(* PLC project TestProject.project, CODESYS CODESYS V3.5 SP16 *)
(* stored: creationDateTime 2020-05-25T13:06:30.288415, modificationDateTime 2020-05-25T13:05:00.4147267 *)

PROGRAM PLC_PRG
  VAR
    mail_arr : ARRAY[1..10] OF STRING := ['Kabanbay', 'Abay', 'Turan', 'Saryarka', 'Pushkina', 'Zeinull', 'Tolegen', 'Hodzhan', 'Zholam', 'Halak'];
    Reader : BarCodeReader;
    i : INT;
  END_VAR

                    IF Start THEN
WHILE TRUE DO
	Timer1(IN:= NOT Timer1.Q AND Start,  PT:=T#2s);
	IF Timer1.Q THEN
		Reader(mail_address:=mail_arr[i]);
		i:=i+1;
	END_IF
END_WHILE
END_IF


                  
END_PROGRAM

FUNCTION_BLOCK BarCodeReader
  VAR_INPUT
    mail_address : STRING;
  END_VAR
  VAR_OUTPUT
    box_num : INT;
  END_VAR
  VAR
    TimerK : TON;
  END_VAR

                    IF  LEFT(mail_address,1)>='A' AND LEFT(mail_address,1)<'F' THEN
	Position_x := 0;
	Position_y := 0;
	IF box1full THEN
		REPEAT
			TimerK(IN:= NOT TimerK.Q,  PT:=T#650MS);
			IF TimerK.Q AND Start THEN
				Position_x:=Position_x+155;
			END_IF
		UNTIL Position_x = 1550
		END_REPEAT
		Position_y:= 150;
		storage:=storage+1;
	ELSE
		REPEAT
			TimerK(IN:= NOT TimerK.Q,  PT:=T#500MS);
			IF TimerK.Q AND Start THEN
				Position_x:=Position_x+67;
			END_IF
		UNTIL Position_x = 335
		END_REPEAT
		Position_y:= 150;
		let1:=let1+1;
	END_IF
	
ELSIF LEFT(mail_address,1)>='F' AND LEFT(mail_address,1)<'K' THEN
	Position_x := 0;
	Position_y := 0;
	IF box2full THEN
		REPEAT
			TimerK(IN:= NOT TimerK.Q,  PT:=T#650MS);
			IF TimerK.Q AND Start THEN
				Position_x:=Position_x+155;
			END_IF
		UNTIL Position_x = 1550
		END_REPEAT
		Position_y:= 150;
		storage:=storage+1;
	ELSE
		REPEAT
			TimerK(IN:= NOT TimerK.Q,  PT:=T#500MS);
			IF TimerK.Q AND Start THEN
				Position_x:=Position_x+55;
			END_IF
		UNTIL Position_x = 550
		END_REPEAT
		Position_y:= 150;
		let2:=let2+1;
	END_IF

ELSIF LEFT(mail_address,1)>='K' AND LEFT(mail_address,1)<'P' THEN
	Position_x := 0;
	Position_y := 0;
	IF box3full THEN
		REPEAT
			TimerK(IN:= NOT TimerK.Q,  PT:=T#650MS);
			IF TimerK.Q AND Start THEN
				Position_x:=Position_x+155;
			END_IF
		UNTIL Position_x = 1550
		END_REPEAT
		Position_y:= 150;
		storage:=storage+1;
	ELSE
		REPEAT
			TimerK(IN:= NOT TimerK.Q,  PT:=T#600MS);
			IF TimerK.Q AND Start THEN
				Position_x:=Position_x+107;
			END_IF
		UNTIL Position_x = 749
		END_REPEAT
		Position_y:= 150;
		let3:=let3+1;
	END_IF

ELSIF LEFT(mail_address,1)>='P' AND LEFT(mail_address,1)<'U' THEN
	Position_x := 0;
	Position_y := 0;
	IF box4full THEN
		REPEAT
			TimerK(IN:= NOT TimerK.Q,  PT:=T#650MS);
			IF TimerK.Q AND Start THEN
				Position_x:=Position_x+155;
			END_IF
		UNTIL Position_x = 1550
		END_REPEAT
		Position_y:= 150;
		storage:=storage+1;
	ELSE
		REPEAT
			TimerK(IN:= NOT TimerK.Q,  PT:=T#1000MS);
			IF TimerK.Q AND Start THEN
				Position_x:=Position_x+97;
			END_IF
		UNTIL Position_x = 970
		END_REPEAT
		Position_y:= 150;
		let4:=let4+1;
	END_IF

ELSIF LEFT(mail_address,1)>='U' AND LEFT(mail_address,1)<='Z' THEN
	Position_x := 0;
	Position_y := 0;
	IF box5full THEN
		REPEAT
			TimerK(IN:= NOT TimerK.Q,  PT:=T#650MS);
			IF TimerK.Q AND Start THEN
				Position_x:=Position_x+155;
			END_IF
		UNTIL Position_x = 1550
		END_REPEAT
		Position_y:= 150;
		storage:=storage+1;
	ELSE
		REPEAT
			TimerK(IN:= NOT TimerK.Q,  PT:=T#1000MS);
			IF TimerK.Q AND Start THEN
				Position_x:=Position_x+119;
			END_IF
		UNTIL Position_x = 1190
		END_REPEAT
		Position_y:= 150;
		let5:=let5+1;
	END_IF
	
END_IF

IF let1 = 3 THEN
	box1full S= TRUE;
ELSIF let2 = 3 THEN
	box2full S= TRUE;
ELSIF let3 = 3 THEN
	box3full S= TRUE;
ELSIF let4 = 3 THEN
	box4full S= TRUE;
ELSIF let5 = 3 THEN
	box5full S= TRUE;
END_IF

                  
END_FUNCTION_BLOCK

CONFIGURATION Device
  RESOURCE Application ON PLC
    VAR_GLOBAL  (* GVL *)
      Start : BOOL;
      Position_x : INT;
      Position_y : INT;
      Timer1 : TON;
      let1 : INT := 0;
      let2 : INT := 0;
      let3 : INT := 0;
      let4 : INT := 0;
      let5 : INT := 0;
      storage : INT := 0;
      box1full : BOOL := FALSE;
      box2full : BOOL := FALSE;
      box3full : BOOL := FALSE;
      box4full : BOOL := FALSE;
      box5full : BOOL := FALSE;
    END_VAR
    TASK MainTask(INTERVAL := T#10ms, PRIORITY := 1);
    TASK VISU_TASK(INTERVAL := T#100ms, PRIORITY := 31);
    PROGRAM PLC_PRG WITH MainTask : PLC_PRG;
    PROGRAM VisuElems.Visu_Prg WITH VISU_TASK : VisuElems.Visu_Prg;
  END_RESOURCE
END_CONFIGURATION
